FUNCTION_BLOCK SerialFB (* rs232_usb *)
  (* Standard: 61499-2 *)
  (* Version 2013_12_09, Gabriel *)
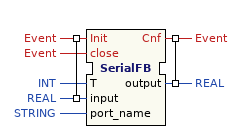
  EVENT_INPUT
    Init WITH input;
    close;
  END_EVENT
  EVENT_OUTPUT
    Cnf WITH output;
  END_EVENT
  VAR_INPUT
    T : INT;
    input : REAL;
    port_name : STRING;
  END_VAR
  VAR_OUTPUT
    output : REAL;
  END_VAR
  SERVICE SerialFB/Serial_Device
    SEQUENCE normal
      SerialFB.Init() -> Serial_Device.init();
      Serial_Device.ok() -> SerialFB.Cnf();
    END_SEQUENCE
  END_SERVICE
END_FUNCTION_BLOCK
